FUNCTION_BLOCK FB_FTP_UploadProgram
VAR_INPUT
	Execute 		: BOOL;
	Username		: STRING;
	Password		: STRING;
	sHost			: STRING;
	sSrcFile		: T_MaxString;
	sDesFile		: T_MaxString;
END_VAR
VAR_OUTPUT
	Busy : BOOL;
	Done : BOOL;
	Error : BOOL;
	ErrorID : DINT;
	ErrorSubID : UDINT;
	Q_tElapsedTime	: TIME;
END_VAR
VAR
	RTRIG_Execute 	: R_TRIG;
	TON_TimeElapsed : TON;
	iState			: DINT := -1;
	i 				: DINT := 0;
	TON_Timeout		: TON;
	fbFTPFileUploadEx: FB_FTP_FileUploadEx;
END_VAR

TON_Timeout(IN := Busy, PT := T#20S);
IF TON_Timeout.Q THEN
	
	iState := 1999;
END_IF

RTRIG_Execute(CLK := Execute);
TON_TimeElapsed(PT:= fbFTPFileUploadEx.tTimeout);
IF(RTRIG_Execute.Q) THEN
	Done 	:= FALSE;
	ErrorID := 0;
	ErrorSubID := 0;
	
	iState 	:= 0;
ELSIF NOT Execute AND NOT Busy THEN
	Busy			:= FALSE;
	Done			:= FALSE;
	Error			:= FALSE;
	
	iState := -1;
END_IF

CASE iState OF
	-1:
		;
	0:
		fbFTPFileUploadEx.bExecute 	:= FALSE;
		TON_TimeElapsed.IN 			:= FALSE;
		Busy 						:= TRUE;
		
		iState 						:= 10;
		
	10:
		fbFTPFileUploadEx.bExecute 	:= TRUE;
		TON_TimeElapsed.IN 			:= TRUE;
		IF(fbFTPFileUploadEx.bBusy) THEN
			iState := 20;
		END_IF
	
	20:	
		IF(NOT fbFTPFileUploadEx.bBusy AND fbFTPFileUploadEx.nProgress = 100) THEN
				
			Q_tElapsedTime := TON_TimeElapsed.ET;
			fbFTPFileUploadEx.bExecute := FALSE;
				
			iState := 999;
		ELSIF(fbFTPFileUploadEx.bError) THEN
			fbFTPFileUploadEx.bExecute := FALSE;
			ErrorSubID := fbFTPFileUploadEx.nErrId;
			
			iState := 1020;
		END_IF
		
	999:
		Done := TRUE;
		Busy := FALSE;
		TON_TimeElapsed.IN := FALSE;
END_CASE

// Error state
IF(iState > 999) THEN
	Busy := FALSE;
	Error := TRUE;
	ErrorID := iState;
ELSE
	Error := FALSE;
	ErrorID := 0;
END_IF

A_Call();

ACTION A_Call:
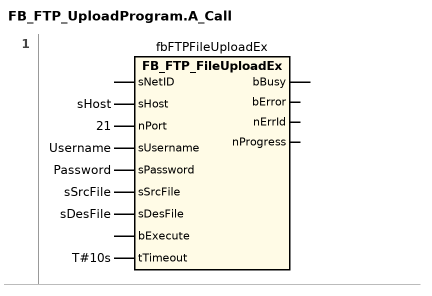
// NETWORK 1
fbFTPFileUploadEx(
    sHost := sHost,
    nPort := 21,
    sUsername := Username,
    sPassword := Password,
    sSrcFile := sSrcFile,
    sDesFile := sDesFile,
    tTimeout := T#10s); // FB_FTP_FileUploadEx
END_ACTION

END_FUNCTION_BLOCK

(* stored: Version 1.1.0.1, ProductVersion 3.1.4024.13
   POU FB_FTP_UploadProgram: Id {8aa173e8-a777-42e1-b51d-8fbacbfec4af}, SpecialFunc None
   Action A_Call: Id {3a76fd94-504d-462b-af0f-71bf6e261682} *)
